FUNCTION_BLOCK _FB_0AC001

VAR_INPUT PERSISTENT

	deviceConfig    : _0AC001_DEV_CONFIG; // Configuration settings for the CT121F device
	
END_VAR
VAR_INPUT 

	  HwToPlc AT %I* : _0AC001_HWTOPLC_PDOS; // Process Data Objects for RWPT01D communication
	
END_VAR
VAR_OUTPUT
	
	analogInput : REAL;
	analogInputRaw : REAL;

END_VAR

_AnalogInputs();

METHOD PRIVATE _AnalogInputs
VAR_INPUT
END_VAR
// Scale sensor distance
analogInput := _Scale(
    X := ((SHL(BYTE_TO_WORD(HwToPlc.inputByte_0),8) OR HwToPlc.inputByte_1)), 
    I_LO := deviceConfig.analogInputLow, 
    I_HI := deviceConfig.analogInputHigh, 
    O_LO := deviceConfig.analogOutputLow, 
    O_HI := deviceConfig.analogOutputHigh
);


// Sensor raw distance
analogInputRaw := (SHL(BYTE_TO_WORD(HwToPlc.inputByte_0),8) OR HwToPlc.inputByte_1);
END_METHOD

METHOD PRIVATE _Scale : REAL
VAR_INPUT
	
	X : REAL;
	I_LO : REAL;
	I_HI : REAL;
	O_LO : REAL;
	O_HI : REAL;
	
END_VAR
IF I_LO = I_HI THEN
	_Scale := O_LO;
ELSE
	_Scale := (O_HI - O_LO) / (I_HI - I_LO) * (LIMIT(I_LO, X, I_HI) - I_LO) + O_LO;
END_IF;
END_METHOD

END_FUNCTION_BLOCK

(* stored: Version 1.1.0.1
   POU _FB_0AC001: Id {c5ec226b-169c-40c7-93b0-61570857e4f3}, SpecialFunc None
   Method _AnalogInputs: Id {1f2b9976-d30d-4584-b1d9-09269ef53957}
   Method _Scale: Id {aa06ca4c-1ac2-48f5-8970-219ce3ccdba7} *)
